// TIA Portal V20 export
// export: Created 2025-12-01T14:57:16.2706351Z, ExportSetting None, DisplayName Totally Integrated Automation Portal, DisplayVersion V20 Update 3, DisplayName TIA Portal Openness, DisplayVersion V20 Update 3, DisplayName TIA Portal Version Control Interface, DisplayVersion V20 Update 3, DisplayName STEP 7 Professional, DisplayVersion V20 Update 3, DisplayName STEP 7 Safety, DisplayVersion V20 Update 2, DisplayName WinCC Basic/Comfort/Advanced, DisplayVersion V20 Update 3, DisplayName WinCC Professional, DisplayVersion V20 Update 3, DisplayName WinCC Unified, DisplayVersion V20 Update 3
DATA_BLOCK "DB841_Recepcion"   // DB841
{ S7_Optimized_Access := 'FALSE' }
AUTHOR : TRACKING
NAME : 20131009
VERSION : 3.1
// stored: AutoNumber false
   VAR
      Mesa { S7_SetPoint := 'True'} : Array[0.."CTE_MaxMesas"] of "UDT_RecepcionDeMesa";   // Array de los Mensajes de Mesas
      DispoArmario { S7_SetPoint := 'True'} : Array[0.."CTE_MaxDispositivos"] of "UDT_RecepcionDeDispositivo";   // Array de los estados de los dispositivos Armarios
      DispoMesa { S7_SetPoint := 'True'} : Array[0.."CTE_MaxMesas"] of "UDT_RecepcionDeDispositivo";   // Array de los estados de los dispositivos Mesas
      DispoMaquina : Array[0.."CTE_MaxMesas"] of "UDT_RecepcionDeDispositivo";   // Array de los estados de los dispositivos Maquina
   END_VAR
BEGIN
END_DATA_BLOCK
